Golden_Tenerife_2026();
Golden_Tenerife_low();
Golden_South_2010();
Golden_Dut1();
Golden_HA_Wrap();
Golden_Near_The_Poles();
Golden_Exact_Poles();
Hour_Angle_Is_Periodic();
Longitude_Is_Periodic();
Outputs_Stay_In_Range();
Round_Trip_Through_RADEC2HADEC();
Inputs_Are_Not_Modified();
Cyclic_Calls_With_Inputs_Set_Once_Are_Stable();

METHOD PRIVATE CheckNear
VAR_INPUT
	fExpected	: LREAL;
	fActual	: LREAL;
	fDelta	: LREAL;
	sName	: STRING(255);
END_VAR
AssertEquals_LREAL(Expected := fExpected, Actual := fActual, Delta := fDelta, Message := sName);
END_METHOD

METHOD PRIVATE CheckAngle
VAR_INPUT
	fExpected	: LREAL;
	fActual	: LREAL;
	fDelta	: LREAL;
	sName	: STRING(255);
END_VAR
VAR
	fDiff	: LREAL;
END_VAR
// angles in degrees, compared modulo 360 so that 359.9999999 and -1.0E-7 are equal
fDiff := fActual - fExpected;
WHILE fDiff > 180.0 DO fDiff := fDiff - 360.0; END_WHILE
WHILE fDiff < -180.0 DO fDiff := fDiff + 360.0; END_WHILE
AssertEquals_LREAL(Expected := 0.0, Actual := fDiff, Delta := fDelta, Message := sName);
END_METHOD

METHOD PRIVATE CheckSeparation
VAR_INPUT
	fLon1	: LREAL;
	fLat1	: LREAL;
	fLon2	: LREAL;
	fLat2	: LREAL;
	fDelta	: LREAL;
	sName	: STRING(255);
END_VAR
VAR
	fD2r	: LREAL;
	fHalfDLat	: LREAL;
	fHalfDLon	: LREAL;
	fHav	: LREAL;
	fSep	: LREAL;
END_VAR
// great-circle separation of two positions (longitude, latitude in degrees) against a tolerance in degrees;
// a difference of longitudes is not a distance on the sky, this is (haversine formula)
fD2r := 0.017453292519943295;
fHalfDLat := (fLat2 - fLat1) * fD2r * 0.5;
fHalfDLon := (fLon2 - fLon1) * fD2r * 0.5;
fHav := SIN(fHalfDLat) * SIN(fHalfDLat) + COS(fLat1 * fD2r) * COS(fLat2 * fD2r) * SIN(fHalfDLon) * SIN(fHalfDLon);
fSep := 2.0 * ASIN(SQRT(LIMIT(0.0, fHav, 1.0))) / fD2r;
AssertEquals_LREAL(Expected := 0.0, Actual := fSep, Delta := fDelta, Message := sName);
END_METHOD

METHOD PRIVATE Golden_Tenerife_2026
VAR
	fb	: AstroBROT.FB_HADEC2RADEC;
END_VAR
TEST('Golden_Tenerife_2026');
fb(jd := 2461300.75, ha := 345.0, dec := 22.01, lon := -16.5, dut1 := 0.0);
CheckAngle(84.28759958479777, fb.ra_out, 1.0E-7, 'Tenerife_2026 ra');
CheckNear(21.993212482320583, fb.dec_out, 1.0E-7, 'Tenerife_2026 dec');
CheckSeparation(84.28749809589803, 21.9932192971722, fb.ra_out, fb.dec_out, 0.0002, 'Tenerife_2026 vs erfa');
TEST_FINISHED();
END_METHOD

METHOD PRIVATE Golden_Tenerife_low
VAR
	fb	: AstroBROT.FB_HADEC2RADEC;
END_VAR
TEST('Golden_Tenerife_low');
fb(jd := 2461300.75, ha := 30.0, dec := -10.0, lon := -16.5, dut1 := 0.0);
CheckAngle(39.36056226713681, fb.ra_out, 1.0E-7, 'Tenerife_low ra');
CheckNear(-10.11975028485237, fb.dec_out, 1.0E-7, 'Tenerife_low dec');
CheckSeparation(39.36047119642502, -10.11974494836338, fb.ra_out, fb.dec_out, 0.0002, 'Tenerife_low vs erfa');
TEST_FINISHED();
END_METHOD

METHOD PRIVATE Golden_South_2010
VAR
	fb	: AstroBROT.FB_HADEC2RADEC;
END_VAR
TEST('Golden_South_2010');
fb(jd := 2455197.5, ha := 100.0, dec := -47.3, lon := -70.7, dut1 := 0.0);
CheckAngle(289.6589544745373, fb.ra_out, 1.0E-7, 'South_2010 ra');
CheckNear(-47.317658585279744, fb.dec_out, 1.0E-7, 'South_2010 dec');
CheckSeparation(289.65896142189746, -47.31759859445048, fb.ra_out, fb.dec_out, 0.0002, 'South_2010 vs erfa');
TEST_FINISHED();
END_METHOD

METHOD PRIVATE Golden_Dut1
VAR
	fb	: AstroBROT.FB_HADEC2RADEC;
END_VAR
TEST('Golden_Dut1');
fb(jd := 2461300.75, ha := 345.0, dec := 22.01, lon := -16.5, dut1 := 0.9);
CheckAngle(84.29135982739001, fb.ra_out, 1.0E-7, 'Tenerife_dut1_plus ra');
CheckNear(21.993222245664892, fb.dec_out, 1.0E-7, 'Tenerife_dut1_plus dec');
CheckSeparation(84.2912582746304, 21.993229060334635, fb.ra_out, fb.dec_out, 0.0002, 'Tenerife_dut1_plus vs erfa');
fb(jd := 2461300.75, ha := 345.0, dec := 22.01, lon := -16.5, dut1 := -0.9);
CheckAngle(84.28383934246425, fb.ra_out, 1.0E-7, 'Tenerife_dut1_minus ra');
CheckNear(21.993202719039957, fb.dec_out, 1.0E-7, 'Tenerife_dut1_minus dec');
CheckSeparation(84.28373791742105, 21.993209534073422, fb.ra_out, fb.dec_out, 0.0002, 'Tenerife_dut1_minus vs erfa');
TEST_FINISHED();
END_METHOD

METHOD PRIVATE Golden_HA_Wrap
VAR
	fb	: AstroBROT.FB_HADEC2RADEC;
END_VAR
TEST('Golden_HA_Wrap');
fb(jd := 2461300.75, ha := 0.0001, dec := 22.01, lon := -16.5, dut1 := 0.0);
CheckAngle(69.28989220623771, fb.ra_out, 1.0E-7, 'HA_wrap_low ra');
CheckNear(21.955213314004528, fb.dec_out, 1.0E-7, 'HA_wrap_low dec');
CheckSeparation(69.28978714407457, 21.95521257782602, fb.ra_out, fb.dec_out, 0.0002, 'HA_wrap_low vs erfa');
fb(jd := 2461300.75, ha := 359.9999, dec := 22.01, lon := -16.5, dut1 := 0.0);
CheckAngle(69.29009214752863, fb.ra_out, 1.0E-7, 'HA_wrap_high ra');
CheckNear(21.95521380223834, fb.dec_out, 1.0E-7, 'HA_wrap_high dec');
CheckSeparation(69.28998708537415, 21.955213066161644, fb.ra_out, fb.dec_out, 0.0002, 'HA_wrap_high vs erfa');
TEST_FINISHED();
END_METHOD

METHOD PRIVATE Golden_Near_The_Poles
VAR
	fb	: AstroBROT.FB_HADEC2RADEC;
END_VAR
TEST('Golden_Near_The_Poles');
fb(jd := 2461300.75, ha := 200.0, dec := 89.9, lon := -16.5, dut1 := 0.0);
CheckAngle(316.7079065490832, fb.ra_out, 1.0E-7, 'Near_north_pole ra');
CheckNear(89.8844737036994, fb.dec_out, 1.0E-7, 'Near_north_pole dec');
CheckSeparation(316.7064081660361, 89.88445978947462, fb.ra_out, fb.dec_out, 0.0002, 'Near_north_pole vs erfa');
fb(jd := 2455197.5, ha := 200.0, dec := -89.9, lon := -70.7, dut1 := 0.0);
CheckAngle(186.30600937346122, fb.ra_out, 1.0E-7, 'Near_south_pole ra');
CheckNear(-89.84872530394176, fb.dec_out, 1.0E-7, 'Near_south_pole dec');
CheckSeparation(186.3367115207879, -89.84875262097749, fb.ra_out, fb.dec_out, 0.0002, 'Near_south_pole vs erfa');
TEST_FINISHED();
END_METHOD

METHOD PRIVATE Golden_Exact_Poles
VAR
	fb	: AstroBROT.FB_HADEC2RADEC;
END_VAR
TEST('Golden_Exact_Poles');
fb(jd := 2461300.75, ha := 200.0, dec := 90.0, lon := -16.5, dut1 := 0.0);
// at exactly dec = +-90 neither ra nor dec is reproducible (d_ra ~ 1/cos(dec) = 1E16, and d_dec is evaluated at that ra), only the bound against erfa is pinned
CheckSeparation(358.71048545509177, 89.85071696591022, fb.ra_out, fb.dec_out, 0.015, 'North_pole vs erfa');
fb(jd := 2455197.5, ha := 200.0, dec := -90.0, lon := -70.7, dut1 := 0.0);
// at exactly dec = +-90 neither ra nor dec is reproducible (d_ra ~ 1/cos(dec) = 1E16, and d_dec is evaluated at that ra), only the bound against erfa is pinned
CheckSeparation(179.80951066897055, -89.94824466951559, fb.ra_out, fb.dec_out, 0.015, 'South_pole vs erfa');
TEST_FINISHED();
END_METHOD

METHOD PRIVATE Hour_Angle_Is_Periodic
VAR
	fb	: AstroBROT.FB_HADEC2RADEC;
END_VAR
TEST('Hour_Angle_Is_Periodic');
// ha and ha +- 360 are the same position; the block does not wrap ra before the corrections, so this also covers the wrap of d_ra (issue #10)
fb(jd := 2461300.75, ha := -15.0, dec := 22.01, lon := -16.5);
CheckAngle(84.28759958479777, fb.ra_out, 1.0E-9, 'ha - 360 ra');
CheckNear(21.993212482320583, fb.dec_out, 1.0E-9, 'ha - 360 dec');
fb(jd := 2461300.75, ha := 705.0, dec := 22.01, lon := -16.5);
CheckAngle(84.28759958479777, fb.ra_out, 1.0E-9, 'ha + 360 ra');
CheckNear(21.993212482320583, fb.dec_out, 1.0E-9, 'ha + 360 dec');
AssertTrue(Condition := fb.ra_out >= 0.0 AND fb.ra_out < 360.0, Message := 'ra_out is within 0 <= ra < 360');
TEST_FINISHED();
END_METHOD

METHOD PRIVATE Longitude_Is_Periodic
VAR
	fb	: AstroBROT.FB_HADEC2RADEC;
END_VAR
TEST('Longitude_Is_Periodic');
fb(jd := 2461300.75, ha := 345.0, dec := 22.01, lon := 343.5);
CheckAngle(84.28759958479777, fb.ra_out, 1.0E-9, 'lon + 360 ra');
fb(jd := 2461300.75, ha := 345.0, dec := 22.01, lon := -376.5);
CheckAngle(84.28759958479777, fb.ra_out, 1.0E-9, 'lon - 360 ra');
TEST_FINISHED();
END_METHOD

METHOD PRIVATE Outputs_Stay_In_Range
VAR
	fb	: AstroBROT.FB_HADEC2RADEC;
	i	: INT;
	fHa	: LREAL;
END_VAR
TEST('Outputs_Stay_In_Range');
FOR i := -1 TO 8 DO
	fHa := 45.0 * i;
	fb(jd := 2461300.75, ha := fHa, dec := 89.9, lon := -16.5);
	AssertTrue(Condition := fb.ra_out >= 0.0 AND fb.ra_out < 360.0 AND fb.dec_out <= 90.0 AND fb.dec_out >= -90.0, Message := 'ha sweep at dec +89.9 stays in range');
	fb(jd := 2461300.75, ha := fHa, dec := -89.9, lon := -16.5);
	AssertTrue(Condition := fb.ra_out >= 0.0 AND fb.ra_out < 360.0 AND fb.dec_out <= 90.0 AND fb.dec_out >= -90.0, Message := 'ha sweep at dec -89.9 stays in range');
	fb(jd := 2461300.75, ha := fHa, dec := 0.0, lon := -16.5);
	AssertTrue(Condition := fb.ra_out >= 0.0 AND fb.ra_out < 360.0 AND fb.dec_out <= 90.0 AND fb.dec_out >= -90.0, Message := 'ha sweep at dec 0 stays in range');
END_FOR
TEST_FINISHED();
END_METHOD

METHOD PRIVATE Round_Trip_Through_RADEC2HADEC
VAR
	fbFwd	: AstroBROT.FB_RADEC2HADEC;
	fbBack	: AstroBROT.FB_HADEC2RADEC;
END_VAR
TEST('Round_Trip_Through_RADEC2HADEC');
// the two blocks are only approximate inverses (nutation and aberration are applied at slightly different
// positions), so 1E-6 deg away from the poles and 2E-4 deg (0.72 arcsec) 0.1 deg from a pole
fbFwd(jd := 2461300.75, ra := 83.63, dec := 22.01, lon := -16.5);
fbBack(jd := 2461300.75, ha := fbFwd.ha_out, dec := fbFwd.dec_out, lon := -16.5);
CheckSeparation(83.63, 22.01, fbBack.ra_out, fbBack.dec_out, 1.0E-6, 'Tenerife_2026');
fbFwd(jd := 2455197.5, ra := 312.5, dec := -47.3, lon := -70.7);
fbBack(jd := 2455197.5, ha := fbFwd.ha_out, dec := fbFwd.dec_out, lon := -70.7);
CheckSeparation(312.5, -47.3, fbBack.ra_out, fbBack.dec_out, 1.0E-6, 'South_2010');
fbFwd(jd := 2461300.75, ra := 359.9999, dec := 22.01, lon := -16.5);
fbBack(jd := 2461300.75, ha := fbFwd.ha_out, dec := fbFwd.dec_out, lon := -16.5);
CheckSeparation(359.9999, 22.01, fbBack.ra_out, fbBack.dec_out, 1.0E-6, 'RA just below 360');
fbFwd(jd := 2461300.75, ra := 0.0001, dec := 22.01, lon := -16.5);
fbBack(jd := 2461300.75, ha := fbFwd.ha_out, dec := fbFwd.dec_out, lon := -16.5);
CheckSeparation(0.0001, 22.01, fbBack.ra_out, fbBack.dec_out, 1.0E-6, 'RA just above 0');
fbFwd(jd := 2461300.75, ra := 200.0, dec := 89.9, lon := -16.5);
fbBack(jd := 2461300.75, ha := fbFwd.ha_out, dec := fbFwd.dec_out, lon := -16.5);
CheckSeparation(200.0, 89.9, fbBack.ra_out, fbBack.dec_out, 0.0002, 'near the north pole');
TEST_FINISHED();
END_METHOD

METHOD PRIVATE Inputs_Are_Not_Modified
VAR
	fb	: AstroBROT.FB_HADEC2RADEC;
END_VAR
TEST('Inputs_Are_Not_Modified');
fb(jd := 2461300.75, ha := 345.0, dec := 22.01, lon := -16.5, dut1 := 0.5);
CheckNear(2461300.75, fb.jd, 0.0, 'jd unchanged');
CheckNear(345.0, fb.ha, 0.0, 'ha unchanged');
CheckNear(22.01, fb.dec, 0.0, 'dec unchanged');
CheckNear(-16.5, fb.lon, 0.0, 'lon unchanged');
CheckNear(0.5, fb.dut1, 0.0, 'dut1 unchanged');
TEST_FINISHED();
END_METHOD

METHOD PRIVATE Cyclic_Calls_With_Inputs_Set_Once_Are_Stable
VAR
	fb	: AstroBROT.FB_HADEC2RADEC;
	i	: INT;
END_VAR
TEST('Cyclic_Calls_With_Inputs_Set_Once_Are_Stable');
fb.jd := 2461300.75;
fb.ha := 345.0;
fb.dec := 22.01;
fb.lon := -16.5;
FOR i := 1 TO 5 DO
	fb();
	CheckAngle(84.28759958479777, fb.ra_out, 1.0E-7, 'cyclic call ra');
	CheckNear(21.993212482320583, fb.dec_out, 1.0E-7, 'cyclic call dec');
END_FOR
TEST_FINISHED();
END_METHOD

END_FUNCTION_BLOCK

// ---- POUs/FB_SUNPOS_Tests.TcPOU
// Tests for AstroBROT.FB_SUNPOS (apparent position of the Sun, port of IDLAstro sunpos.pro).
//
// GENERATED by AstroBROT/testing/gen_block_tests.py from testing/golden_blocks.py, do not edit the numbers by hand.
// Golden values from the Python port of the ST (1E-7 deg). Independently of the port the position is compared with a
// position built from erfa (epv00 / pmat06 / nut06a): 1.5E-3 deg = 5.4 arcsec, the measured maximum is 3.2 arcsec and
// the IDLAstro documentation states 7.3 arcsec for 1900-2100. The last tests are plain sanity checks (equinox,
// solstice, obliquity, RA rate) that need neither the port nor erfa.
FUNCTION_BLOCK FB_SUNPOS_Tests EXTENDS TcUnit.FB_TestSuite
VAR
END_VAR

Golden_Epoch_1900_And_J2000();
Golden_Start_2010();
Golden_Tenerife_2026();
Golden_Year_2050();
Golden_Equinox_And_Solstice_2026();
Sanity_Equinox_Solstice_Obliquity();
Sanity_Right_Ascension_Advances_About_One_Degree_Per_Day();
Inputs_Are_Not_Modified();
Cyclic_Calls_With_Inputs_Set_Once_Are_Stable();

METHOD PRIVATE CheckNear
VAR_INPUT
	fExpected	: LREAL;
	fActual	: LREAL;
	fDelta	: LREAL;
	sName	: STRING(255);
END_VAR
AssertEquals_LREAL(Expected := fExpected, Actual := fActual, Delta := fDelta, Message := sName);
END_METHOD

METHOD PRIVATE CheckAngle
VAR_INPUT
	fExpected	: LREAL;
	fActual	: LREAL;
	fDelta	: LREAL;
	sName	: STRING(255);
END_VAR
VAR
	fDiff	: LREAL;
END_VAR
// angles in degrees, compared modulo 360 so that 359.9999999 and -1.0E-7 are equal
fDiff := fActual - fExpected;
WHILE fDiff > 180.0 DO fDiff := fDiff - 360.0; END_WHILE
WHILE fDiff < -180.0 DO fDiff := fDiff + 360.0; END_WHILE
AssertEquals_LREAL(Expected := 0.0, Actual := fDiff, Delta := fDelta, Message := sName);
END_METHOD

METHOD PRIVATE CheckSeparation
VAR_INPUT
	fLon1	: LREAL;
	fLat1	: LREAL;
	fLon2	: LREAL;
	fLat2	: LREAL;
	fDelta	: LREAL;
	sName	: STRING(255);
END_VAR
VAR
	fD2r	: LREAL;
	fHalfDLat	: LREAL;
	fHalfDLon	: LREAL;
	fHav	: LREAL;
	fSep	: LREAL;
END_VAR
// great-circle separation of two positions (longitude, latitude in degrees) against a tolerance in degrees;
// a difference of longitudes is not a distance on the sky, this is (haversine formula)
fD2r := 0.017453292519943295;
fHalfDLat := (fLat2 - fLat1) * fD2r * 0.5;
fHalfDLon := (fLon2 - fLon1) * fD2r * 0.5;
fHav := SIN(fHalfDLat) * SIN(fHalfDLat) + COS(fLat1 * fD2r) * COS(fLat2 * fD2r) * SIN(fHalfDLon) * SIN(fHalfDLon);
fSep := 2.0 * ASIN(SQRT(LIMIT(0.0, fHav, 1.0))) / fD2r;
AssertEquals_LREAL(Expected := 0.0, Actual := fSep, Delta := fDelta, Message := sName);
END_METHOD

METHOD PRIVATE Golden_Epoch_1900_And_J2000
VAR
	fb	: AstroBROT.FB_SUNPOS;
END_VAR
TEST('Golden_Epoch_1900_And_J2000');
fb(jd := 2415020.0);
CheckAngle(280.4932027906667, fb.ra, 1.0E-7, 'Epoch_1900 ra');
CheckNear(-23.1010537507843, fb.dec, 1.0E-7, 'Epoch_1900 dec');
CheckNear(279.6444003923051, fb.longmed, 1.0E-7, 'Epoch_1900 longmed');
CheckNear(23.451814403891508, fb.oblt, 1.0E-7, 'Epoch_1900 oblt');
CheckSeparation(280.49336588705194, -23.100882447052207, fb.ra, fb.dec, 0.0015, 'Epoch_1900 vs erfa');
fb(jd := 2451545.0);
CheckAngle(281.27675114506104, fb.ra, 1.0E-7, 'J2000 ra');
CheckNear(-23.03291144063576, fb.dec, 1.0E-7, 'J2000 dec');
CheckNear(280.37698786565545, fb.longmed, 1.0E-7, 'J2000 longmed');
CheckNear(23.437814186179185, fb.oblt, 1.0E-7, 'J2000 oblt');
CheckSeparation(281.2776898567173, -23.032708521099703, fb.ra, fb.dec, 0.0015, 'J2000 vs erfa');
TEST_FINISHED();
END_METHOD

METHOD PRIVATE Golden_Start_2010
VAR
	fb	: AstroBROT.FB_SUNPOS;
END_VAR
TEST('Golden_Start_2010');
fb(jd := 2455197.5);
CheckAngle(281.36670259981736, fb.ra, 1.0E-7, 'Start_2010 ra');
CheckNear(-23.027520406003863, fb.dec, 1.0E-7, 'Start_2010 dec');
CheckNear(280.4515850797381, fb.longmed, 1.0E-7, 'Start_2010 longmed');
CheckNear(23.438922135094707, fb.oblt, 1.0E-7, 'Start_2010 oblt');
CheckSeparation(281.3668435021951, -23.027353107638568, fb.ra, fb.dec, 0.0015, 'Start_2010 vs erfa');
TEST_FINISHED();
END_METHOD

METHOD PRIVATE Golden_Tenerife_2026
VAR
	fb	: AstroBROT.FB_SUNPOS;
END_VAR
TEST('Golden_Tenerife_2026');
fb(jd := 2461300.75);
CheckAngle(174.8393337772982, fb.ra, 1.0E-7, 'Tenerife_2026 ra');
CheckNear(2.2331274030840897, fb.dec, 1.0E-7, 'Tenerife_2026 dec');
CheckNear(174.38128640738705, fb.longmed, 1.0E-7, 'Tenerife_2026 longmed');
CheckNear(23.437983366242445, fb.oblt, 1.0E-7, 'Tenerife_2026 oblt');
CheckSeparation(174.84005201634432, 2.232830546071217, fb.ra, fb.dec, 0.0015, 'Tenerife_2026 vs erfa');
TEST_FINISHED();
END_METHOD

METHOD PRIVATE Golden_Year_2050
VAR
	fb	: AstroBROT.FB_SUNPOS;
END_VAR
TEST('Golden_Year_2050');
fb(jd := 2469807.5);
CheckAngle(281.68738605381645, fb.ra, 1.0E-7, 'Year_2050 ra');
CheckNear(-22.996590225692305, fb.dec, 1.0E-7, 'Year_2050 dec');
CheckNear(280.748664812077, fb.longmed, 1.0E-7, 'Year_2050 longmed');
CheckNear(23.431419887249728, fb.oblt, 1.0E-7, 'Year_2050 oblt');
CheckSeparation(281.6880601925095, -22.996415910571415, fb.ra, fb.dec, 0.0015, 'Year_2050 vs erfa');
TEST_FINISHED();
END_METHOD

METHOD PRIVATE Golden_Equinox_And_Solstice_2026
VAR
	fb	: AstroBROT.FB_SUNPOS;
END_VAR
TEST('Golden_Equinox_And_Solstice_2026');
fb(jd := 2461120.5);
CheckAngle(0.3503559250411667, fb.ra, 1.0E-7, 'March_equinox_2026 ra');
CheckNear(0.15188894029624206, fb.dec, 1.0E-7, 'March_equinox_2026 dec');
CheckNear(0.3857660381664108, fb.longmed, 1.0E-7, 'March_equinox_2026 longmed');
CheckNear(23.438239257244735, fb.oblt, 1.0E-7, 'March_equinox_2026 oblt');
CheckSeparation(0.35013805050580776, 0.15179565874940165, fb.ra, fb.dec, 0.0015, 'March_equinox_2026 vs erfa');
fb(jd := 2461212.5);
CheckAngle(89.63389115907498, fb.ra, 1.0E-7, 'June_solstice_2026 ra');
CheckNear(23.437689690338015, fb.dec, 1.0E-7, 'June_solstice_2026 dec');
CheckNear(89.66763149502222, fb.longmed, 1.0E-7, 'June_solstice_2026 longmed');
CheckNear(23.43811655330089, fb.oblt, 1.0E-7, 'June_solstice_2026 oblt');
CheckSeparation(89.63460394632473, 23.437550528896672, fb.ra, fb.dec, 0.0015, 'June_solstice_2026 vs erfa');
TEST_FINISHED();
END_METHOD

METHOD PRIVATE Sanity_Equinox_Solstice_Obliquity
VAR
	fb	: AstroBROT.FB_SUNPOS;
END_VAR
TEST('Sanity_Equinox_Solstice_Obliquity');
// 2026-03-21 00:00 UT is 9 h after the March equinox: the Sun is at RA about 0.35 deg, Dec about +0.15 deg
fb(jd := 2461120.5);
CheckAngle(0.35, fb.ra, 0.3, 'March equinox ra');
CheckNear(0.15, fb.dec, 0.1, 'March equinox dec');
// 2026-06-21 00:00 UT is 8 h before the June solstice: Dec is at its maximum, RA about 89.6 deg
fb(jd := 2461212.5);
CheckNear(23.44, fb.dec, 0.02, 'June solstice dec');
CheckAngle(89.6, fb.ra, 0.3, 'June solstice ra');
// true obliquity of the ecliptic in 2026
CheckNear(23.437, fb.oblt, 0.005, 'oblt 2026');
TEST_FINISHED();
END_METHOD

METHOD PRIVATE Sanity_Right_Ascension_Advances_About_One_Degree_Per_Day
VAR
	fb	: AstroBROT.FB_SUNPOS;
	fbNext	: AstroBROT.FB_SUNPOS;
	i	: INT;
	fStep	: LREAL;
END_VAR
TEST('Sanity_Right_Ascension_Advances_About_One_Degree_Per_Day');
// over a year the daily change of RA is between 0.85 and 1.15 deg (0.91 to 1.11 in reality); this also crosses the wrap at 360
FOR i := 0 TO 36 DO
	fb(jd := 2461041.5 + 10.0 * i);
	fbNext(jd := 2461042.5 + 10.0 * i);
	fStep := fbNext.ra - fb.ra;
	IF fStep < 0.0 THEN fStep := fStep + 360.0; END_IF
	AssertTrue(Condition := fStep > 0.85 AND fStep < 1.15, Message := 'daily RA step within 0.85 .. 1.15 deg');
	AssertTrue(Condition := fb.ra >= 0.0 AND fb.ra < 360.0 AND ABS(fb.dec) < 23.5, Message := 'ra in range, |dec| below the obliquity');
END_FOR
TEST_FINISHED();
END_METHOD

METHOD PRIVATE Inputs_Are_Not_Modified
VAR
	fb	: AstroBROT.FB_SUNPOS;
END_VAR
TEST('Inputs_Are_Not_Modified');
fb(jd := 2461300.75);
CheckNear(2461300.75, fb.jd, 0.0, 'jd unchanged');
TEST_FINISHED();
END_METHOD

METHOD PRIVATE Cyclic_Calls_With_Inputs_Set_Once_Are_Stable
VAR
	fb	: AstroBROT.FB_SUNPOS;
	i	: INT;
END_VAR
TEST('Cyclic_Calls_With_Inputs_Set_Once_Are_Stable');
fb.jd := 2461300.75;
FOR i := 1 TO 5 DO
	fb();
	CheckAngle(174.8393337772982, fb.ra, 1.0E-7, 'cyclic call ra');
	CheckNear(2.2331274030840897, fb.dec, 1.0E-7, 'cyclic call dec');
END_FOR
TEST_FINISHED();
END_METHOD

END_FUNCTION_BLOCK

// ---- POUs/FB_EdgeCases_Tests.TcPOU
// Edge cases of FB_EQ2HOR and FB_HOR2EQ: the celestial poles, an observer at a pole and on the equator, the zenith and
// the nadir, wrap-around of RA and azimuth, positions below the horizon and out-of-range angles.
//
// GENERATED by AstroBROT/testing/gen_block_tests.py from testing/golden_blocks.py, do not edit the numbers by hand.
// Every golden case is checked against the Python port of the ST (1E-7 deg) and against erfa (atco13 / atoc13) as a
// great-circle separation (2E-4 deg = 0.72 arcsec, no refraction, dut1 = 0). Altitude and azimuth are compared as a
// separation on the sky, not as two separate angle differences: near the zenith an azimuth difference is amplified by
// 1 / cos(alt) and says little about the pointing error (Azimuth_Difference_Is_Not_A_Sky_Separation).
FUNCTION_BLOCK FB_EdgeCases_Tests EXTENDS TcUnit.FB_TestSuite
VAR
END_VAR

EQ2HOR_North_celestial_pole();
EQ2HOR_South_celestial_pole();
EQ2HOR_RA_wrap_low();
EQ2HOR_RA_wrap_high();
EQ2HOR_Below_horizon();
EQ2HOR_Observer_at_north_pole();
EQ2HOR_Observer_at_south_pole();
EQ2HOR_Observer_on_equator();
HOR2EQ_Zenith_az0();
HOR2EQ_Zenith_az180();
HOR2EQ_Nadir();
HOR2EQ_Horizon_north();
HOR2EQ_Az_wrap_low();
HOR2EQ_Az_wrap_high();
HOR2EQ_Observer_at_north_pole();
HOR2EQ_Observer_at_south_pole();
HOR2EQ_Observer_on_equator();
HOR2EQ_Azimuth_Does_Not_Matter_At_The_Zenith();
HOR2EQ_Azimuth_Is_Periodic();
EQ2HOR_Right_Ascension_Is_Periodic();
EQ2HOR_Longitude_Is_Periodic();
EQ2HOR_Outputs_Stay_In_Range();
HOR2EQ_Outputs_Stay_In_Range();
Azimuth_Difference_Is_Not_A_Sky_Separation();

METHOD PRIVATE CheckNear
VAR_INPUT
	fExpected	: LREAL;
	fActual	: LREAL;
	fDelta	: LREAL;
	sName	: STRING(255);
END_VAR
AssertEquals_LREAL(Expected := fExpected, Actual := fActual, Delta := fDelta, Message := sName);
END_METHOD

METHOD PRIVATE CheckAngle
VAR_INPUT
	fExpected	: LREAL;
	fActual	: LREAL;
	fDelta	: LREAL;
	sName	: STRING(255);
END_VAR
VAR
	fDiff	: LREAL;
END_VAR
// angles in degrees, compared modulo 360 so that 359.9999999 and -1.0E-7 are equal
fDiff := fActual - fExpected;
WHILE fDiff > 180.0 DO fDiff := fDiff - 360.0; END_WHILE
WHILE fDiff < -180.0 DO fDiff := fDiff + 360.0; END_WHILE
AssertEquals_LREAL(Expected := 0.0, Actual := fDiff, Delta := fDelta, Message := sName);
END_METHOD

METHOD PRIVATE CheckSeparation
VAR_INPUT
	fLon1	: LREAL;
	fLat1	: LREAL;
	fLon2	: LREAL;
	fLat2	: LREAL;
	fDelta	: LREAL;
	sName	: STRING(255);
END_VAR
VAR
	fD2r	: LREAL;
	fHalfDLat	: LREAL;
	fHalfDLon	: LREAL;
	fHav	: LREAL;
	fSep	: LREAL;
END_VAR
// great-circle separation of two positions (longitude, latitude in degrees) against a tolerance in degrees;
// a difference of longitudes is not a distance on the sky, this is (haversine formula)
fD2r := 0.017453292519943295;
fHalfDLat := (fLat2 - fLat1) * fD2r * 0.5;
fHalfDLon := (fLon2 - fLon1) * fD2r * 0.5;
fHav := SIN(fHalfDLat) * SIN(fHalfDLat) + COS(fLat1 * fD2r) * COS(fLat2 * fD2r) * SIN(fHalfDLon) * SIN(fHalfDLon);
fSep := 2.0 * ASIN(SQRT(LIMIT(0.0, fHav, 1.0))) / fD2r;
AssertEquals_LREAL(Expected := 0.0, Actual := fSep, Delta := fDelta, Message := sName);
END_METHOD

METHOD PRIVATE EQ2HOR_North_celestial_pole
VAR
	fb	: AstroBROT.FB_EQ2HOR;
END_VAR
TEST('EQ2HOR_North_celestial_pole');
fb(ra := 0.0, dec := 90.0, jd := 2461300.75, lon := -16.5, lat := 28.3, refract := FALSE);
CheckNear(28.250439967419368, fb.alt, 1.0E-7, 'North_celestial_pole alt');
CheckAngle(0.15978772490399448, fb.az, 1.0E-7, 'North_celestial_pole az');
CheckSeparation(0.159877225222193, 28.250414281534653, fb.az, fb.alt, 0.0002, 'North_celestial_pole vs erfa');
TEST_FINISHED();
END_METHOD

METHOD PRIVATE EQ2HOR_South_celestial_pole
VAR
	fb	: AstroBROT.FB_EQ2HOR;
END_VAR
TEST('EQ2HOR_South_celestial_pole');
fb(ra := 0.0, dec := -90.0, jd := 2455197.5, lon := -70.7, lat := -30.2, refract := FALSE);
CheckNear(30.24486015624291, fb.alt, 1.0E-7, 'South_celestial_pole alt');
CheckAngle(180.02996665539834, fb.az, 1.0E-7, 'South_celestial_pole az');
CheckSeparation(180.02986430898196, 30.244862822992012, fb.az, fb.alt, 0.0002, 'South_celestial_pole vs erfa');
TEST_FINISHED();
END_METHOD

METHOD PRIVATE EQ2HOR_RA_wrap_low
VAR
	fb	: AstroBROT.FB_EQ2HOR;
END_VAR
TEST('EQ2HOR_RA_wrap_low');
fb(ra := 0.0001, dec := 22.01, jd := 2461300.75, lon := -16.5, lat := 28.3, refract := FALSE);
CheckNear(27.80734764100336, fb.alt, 1.0E-7, 'RA_wrap_low alt');
CheckAngle(281.5592750159755, fb.az, 1.0E-7, 'RA_wrap_low az');
CheckSeparation(281.55928456225905, 27.807403036183125, fb.az, fb.alt, 0.0002, 'RA_wrap_low vs erfa');
TEST_FINISHED();
END_METHOD

METHOD PRIVATE EQ2HOR_RA_wrap_high
VAR
	fb	: AstroBROT.FB_EQ2HOR;
END_VAR
TEST('EQ2HOR_RA_wrap_high');
fb(ra := 359.9999, dec := 22.01, jd := 2461300.75, lon := -16.5, lat := 28.3, refract := FALSE);
CheckNear(27.807174935931986, fb.alt, 1.0E-7, 'RA_wrap_high alt');
CheckAngle(281.55935130398774, fb.az, 1.0E-7, 'RA_wrap_high az');
CheckSeparation(281.5593608503559, 27.80723033089579, fb.az, fb.alt, 0.0002, 'RA_wrap_high vs erfa');
TEST_FINISHED();
END_METHOD

METHOD PRIVATE EQ2HOR_Below_horizon
VAR
	fb	: AstroBROT.FB_EQ2HOR;
END_VAR
TEST('EQ2HOR_Below_horizon');
fb(ra := 200.0, dec := -60.0, jd := 2461300.75, lon := -16.5, lat := 28.3, refract := FALSE);
CheckNear(-44.20054793244784, fb.alt, 1.0E-7, 'Below_horizon alt');
CheckAngle(148.24726062401623, fb.az, 1.0E-7, 'Below_horizon az');
CheckSeparation(148.2471745159021, -44.20052670358075, fb.az, fb.alt, 0.0002, 'Below_horizon vs erfa');
TEST_FINISHED();
END_METHOD

METHOD PRIVATE EQ2HOR_Observer_at_north_pole
VAR
	fb	: AstroBROT.FB_EQ2HOR;
END_VAR
TEST('EQ2HOR_Observer_at_north_pole');
fb(ra := 83.63, dec := 22.01, jd := 2461300.75, lon := 0.0, lat := 90.0, refract := FALSE);
CheckNear(22.028492329681235, fb.alt, 1.0E-7, 'Observer_at_north_pole alt');
CheckAngle(182.15756303104874, fb.az, 1.0E-7, 'Observer_at_north_pole az');
CheckSeparation(182.15754329791073, 22.028492563126676, fb.az, fb.alt, 0.0002, 'Observer_at_north_pole vs erfa');
TEST_FINISHED();
END_METHOD

METHOD PRIVATE EQ2HOR_Observer_at_south_pole
VAR
	fb	: AstroBROT.FB_EQ2HOR;
END_VAR
TEST('EQ2HOR_Observer_at_south_pole');
fb(ra := 83.63, dec := -22.01, jd := 2461300.75, lon := 0.0, lat := -90.0, refract := FALSE);
CheckNear(21.987455170067353, fb.alt, 1.0E-7, 'Observer_at_south_pole alt');
CheckAngle(357.7223600600331, fb.az, 1.0E-7, 'Observer_at_south_pole az');
CheckSeparation(357.7223798312026, 21.987453746489294, fb.az, fb.alt, 0.0002, 'Observer_at_south_pole vs erfa');
TEST_FINISHED();
END_METHOD

METHOD PRIVATE EQ2HOR_Observer_on_equator
VAR
	fb	: AstroBROT.FB_EQ2HOR;
END_VAR
TEST('EQ2HOR_Observer_on_equator');
fb(ra := 83.63, dec := 22.01, jd := 2461300.75, lon := -16.5, lat := 0.0, refract := FALSE);
CheckNear(63.91012183292501, fb.alt, 1.0E-7, 'Observer_on_equator alt');
CheckAngle(31.47678113024893, fb.az, 1.0E-7, 'Observer_on_equator az');
CheckSeparation(31.476987570998272, 63.910069653766755, fb.az, fb.alt, 0.0002, 'Observer_on_equator vs erfa');
TEST_FINISHED();
END_METHOD

METHOD PRIVATE HOR2EQ_Zenith_az0
VAR
	fb	: AstroBROT.FB_HOR2EQ;
END_VAR
TEST('HOR2EQ_Zenith_az0');
fb(alt := 90.0, az := 0.0, jd := 2461300.75, lon := -16.5, lat := 28.3, refract := FALSE);
CheckAngle(69.27121990661907, fb.ra, 1.0E-7, 'Zenith_az0 ra');
CheckNear(28.245793686130707, fb.dec, 1.0E-7, 'Zenith_az0 dec');
CheckSeparation(69.27111043655914, 28.245793175984534, fb.ra, fb.dec, 0.0002, 'Zenith_az0 vs erfa');
TEST_FINISHED();
END_METHOD

METHOD PRIVATE HOR2EQ_Zenith_az180
VAR
	fb	: AstroBROT.FB_HOR2EQ;
END_VAR
TEST('HOR2EQ_Zenith_az180');
fb(alt := 90.0, az := 180.0, jd := 2461300.75, lon := -16.5, lat := 28.3, refract := FALSE);
CheckAngle(69.27121990661907, fb.ra, 1.0E-7, 'Zenith_az180 ra');
CheckNear(28.245793686130707, fb.dec, 1.0E-7, 'Zenith_az180 dec');
CheckSeparation(69.27111043655914, 28.245793175984534, fb.ra, fb.dec, 0.0002, 'Zenith_az180 vs erfa');
TEST_FINISHED();
END_METHOD

METHOD PRIVATE HOR2EQ_Nadir
VAR
	fb	: AstroBROT.FB_HOR2EQ;
END_VAR
TEST('HOR2EQ_Nadir');
fb(alt := -90.0, az := 0.0, jd := 2461300.75, lon := -16.5, lat := 28.3, refract := FALSE);
CheckAngle(249.2743126674054, fb.ra, 1.0E-7, 'Nadir ra');
CheckNear(-28.244996713786396, fb.dec, 1.0E-7, 'Nadir dec');
CheckSeparation(249.27437964349747, -28.24499592575831, fb.ra, fb.dec, 0.0002, 'Nadir vs erfa');
TEST_FINISHED();
END_METHOD

METHOD PRIVATE HOR2EQ_Horizon_north
VAR
	fb	: AstroBROT.FB_HOR2EQ;
END_VAR
TEST('HOR2EQ_Horizon_north');
fb(alt := 0.0, az := 0.0, jd := 2461300.75, lon := -16.5, lat := 28.3, refract := FALSE);
CheckAngle(249.60995502319435, fb.ra, 1.0E-7, 'Horizon_north ra');
CheckNear(61.7487089558397, fb.dec, 1.0E-7, 'Horizon_north dec');
CheckSeparation(249.61009729239348, 61.74870711776769, fb.ra, fb.dec, 0.0002, 'Horizon_north vs erfa');
TEST_FINISHED();
END_METHOD

METHOD PRIVATE HOR2EQ_Az_wrap_low
VAR
	fb	: AstroBROT.FB_HOR2EQ;
END_VAR
TEST('HOR2EQ_Az_wrap_low');
fb(alt := 45.0, az := 0.0001, jd := 2461300.75, lon := -16.5, lat := 28.3, refract := FALSE);
CheckAngle(68.88002145549598, fb.ra, 1.0E-7, 'Az_wrap_low ra');
CheckNear(73.24907291497094, fb.dec, 1.0E-7, 'Az_wrap_low dec');
CheckSeparation(68.8797303761049, 73.24907332545713, fb.ra, fb.dec, 0.0002, 'Az_wrap_low vs erfa');
TEST_FINISHED();
END_METHOD

METHOD PRIVATE HOR2EQ_Az_wrap_high
VAR
	fb	: AstroBROT.FB_HOR2EQ;
END_VAR
TEST('HOR2EQ_Az_wrap_high');
fb(alt := 45.0, az := 359.9999, jd := 2461300.75, lon := -16.5, lat := 28.3, refract := FALSE);
CheckAngle(68.87953075699878, fb.ra, 1.0E-7, 'Az_wrap_high ra');
CheckNear(73.24907170989893, fb.dec, 1.0E-7, 'Az_wrap_high dec');
CheckSeparation(68.87923967758073, 73.2490721197454, fb.ra, fb.dec, 0.0002, 'Az_wrap_high vs erfa');
TEST_FINISHED();
END_METHOD

METHOD PRIVATE HOR2EQ_Observer_at_north_pole
VAR
	fb	: AstroBROT.FB_HOR2EQ;
END_VAR
TEST('HOR2EQ_Observer_at_north_pole');
fb(alt := 40.0, az := 100.0, jd := 2461300.75, lon := 0.0, lat := 90.0, refract := FALSE);
CheckAngle(165.82212182028053, fb.ra, 1.0E-7, 'Observer_at_north_pole ra');
CheckNear(40.14345354944047, fb.dec, 1.0E-7, 'Observer_at_north_pole dec');
CheckSeparation(165.82210357343894, 40.14345009010985, fb.ra, fb.dec, 0.0002, 'Observer_at_north_pole vs erfa');
TEST_FINISHED();
END_METHOD

METHOD PRIVATE HOR2EQ_Observer_at_south_pole
VAR
	fb	: AstroBROT.FB_HOR2EQ;
END_VAR
TEST('HOR2EQ_Observer_at_south_pole');
fb(alt := -20.0, az := 100.0, jd := 2461300.75, lon := 0.0, lat := -90.0, refract := FALSE);
CheckAngle(185.85805478189764, fb.ra, 1.0E-7, 'Observer_at_south_pole ra');
CheckNear(20.14661753333691, fb.dec, 1.0E-7, 'Observer_at_south_pole dec');
CheckSeparation(185.85803179512064, 20.146612025652036, fb.ra, fb.dec, 0.0002, 'Observer_at_south_pole vs erfa');
TEST_FINISHED();
END_METHOD

METHOD PRIVATE HOR2EQ_Observer_on_equator
VAR
	fb	: AstroBROT.FB_HOR2EQ;
END_VAR
TEST('HOR2EQ_Observer_on_equator');
fb(alt := 60.0, az := 250.0, jd := 2461300.75, lon := -16.5, lat := 0.0, refract := FALSE);
CheckAngle(40.87970090453398, fb.ra, 1.0E-7, 'Observer_on_equator ra');
CheckNear(-9.963791072363595, fb.dec, 1.0E-7, 'Observer_on_equator dec');
CheckSeparation(40.879599464361846, -9.963785329026702, fb.ra, fb.dec, 0.0002, 'Observer_on_equator vs erfa');
TEST_FINISHED();
END_METHOD

METHOD PRIVATE HOR2EQ_Azimuth_Does_Not_Matter_At_The_Zenith
VAR
	fbA	: AstroBROT.FB_HOR2EQ;
	fbB	: AstroBROT.FB_HOR2EQ;
END_VAR
TEST('HOR2EQ_Azimuth_Does_Not_Matter_At_The_Zenith');
fbA(alt := 90.0, az := 0.0, jd := 2461300.75, lon := -16.5, lat := 28.3, refract := FALSE);
fbB(alt := 90.0, az := 180.0, jd := 2461300.75, lon := -16.5, lat := 28.3, refract := FALSE);
CheckAngle(fbA.ra, fbB.ra, 1.0E-9, 'ra');
CheckNear(fbA.dec, fbB.dec, 1.0E-9, 'dec');
AssertTrue(Condition := fbA.dec > 0.0 AND fbA.dec < 90.0, Message := 'the zenith of a northern site has 0 < dec < 90 (no NaN from ASIN)');
TEST_FINISHED();
END_METHOD

METHOD PRIVATE HOR2EQ_Azimuth_Is_Periodic
VAR
	fbRef	: AstroBROT.FB_HOR2EQ;
	fb	: AstroBROT.FB_HOR2EQ;
END_VAR
TEST('HOR2EQ_Azimuth_Is_Periodic');
fbRef(alt := 45.0, az := 350.0, jd := 2461300.75, lon := -16.5, lat := 28.3, refract := FALSE);
fb(alt := 45.0, az := -10.0, jd := 2461300.75, lon := -16.5, lat := 28.3, refract := FALSE);
CheckAngle(fbRef.ra, fb.ra, 1.0E-9, 'az -10 ra');
CheckNear(fbRef.dec, fb.dec, 1.0E-9, 'az -10 dec');
fb(alt := 45.0, az := 710.0, jd := 2461300.75, lon := -16.5, lat := 28.3, refract := FALSE);
CheckAngle(fbRef.ra, fb.ra, 1.0E-9, 'az 710 ra');
CheckNear(fbRef.dec, fb.dec, 1.0E-9, 'az 710 dec');
TEST_FINISHED();
END_METHOD

METHOD PRIVATE EQ2HOR_Right_Ascension_Is_Periodic
VAR
	fbRef	: AstroBROT.FB_EQ2HOR;
	fb	: AstroBROT.FB_EQ2HOR;
END_VAR
TEST('EQ2HOR_Right_Ascension_Is_Periodic');
fbRef(ra := 83.63, dec := 22.01, jd := 2461300.75, lon := -16.5, lat := 28.3, refract := FALSE);
fb(ra := -276.37, dec := 22.01, jd := 2461300.75, lon := -16.5, lat := 28.3, refract := FALSE);
CheckNear(fbRef.alt, fb.alt, 1.0E-9, 'ra -276.37 alt');
CheckAngle(fbRef.az, fb.az, 1.0E-9, 'ra -276.37 az');
fb(ra := 443.63, dec := 22.01, jd := 2461300.75, lon := -16.5, lat := 28.3, refract := FALSE);
CheckNear(fbRef.alt, fb.alt, 1.0E-9, 'ra 443.63 alt');
CheckAngle(fbRef.az, fb.az, 1.0E-9, 'ra 443.63 az');
TEST_FINISHED();
END_METHOD

METHOD PRIVATE EQ2HOR_Longitude_Is_Periodic
VAR
	fbRef	: AstroBROT.FB_EQ2HOR;
	fb	: AstroBROT.FB_EQ2HOR;
END_VAR
TEST('EQ2HOR_Longitude_Is_Periodic');
fbRef(ra := 83.63, dec := 22.01, jd := 2461300.75, lon := -16.5, lat := 28.3, refract := FALSE);
fb(ra := 83.63, dec := 22.01, jd := 2461300.75, lon := 343.5, lat := 28.3, refract := FALSE);
CheckNear(fbRef.alt, fb.alt, 1.0E-9, 'lon 343.5 alt');
CheckAngle(fbRef.az, fb.az, 1.0E-9, 'lon 343.5 az');
TEST_FINISHED();
END_METHOD

METHOD PRIVATE EQ2HOR_Outputs_Stay_In_Range
VAR
	fb	: AstroBROT.FB_EQ2HOR;
	i	: INT;
	fDec	: LREAL;
END_VAR
TEST('EQ2HOR_Outputs_Stay_In_Range');
// declinations from pole to pole for observers at both poles, on the equator and at a mid latitude
FOR i := -2 TO 2 DO
	fDec := 45.0 * i;
	fb(ra := 200.0, dec := fDec, jd := 2461300.75, lon := 0.0, lat := 90.0, refract := FALSE);
	AssertTrue(Condition := fb.alt >= -90.0 AND fb.alt <= 90.0 AND fb.az >= 0.0 AND fb.az <= 360.0, Message := 'observer at the north pole');
	fb(ra := 200.0, dec := fDec, jd := 2461300.75, lon := 0.0, lat := -90.0, refract := FALSE);
	AssertTrue(Condition := fb.alt >= -90.0 AND fb.alt <= 90.0 AND fb.az >= 0.0 AND fb.az <= 360.0, Message := 'observer at the south pole');
	fb(ra := 200.0, dec := fDec, jd := 2461300.75, lon := 0.0, lat := 0.0, refract := FALSE);
	AssertTrue(Condition := fb.alt >= -90.0 AND fb.alt <= 90.0 AND fb.az >= 0.0 AND fb.az <= 360.0, Message := 'observer on the equator');
	fb(ra := 200.0, dec := fDec, jd := 2461300.75, lon := -16.5, lat := 28.3, refract := FALSE);
	AssertTrue(Condition := fb.alt >= -90.0 AND fb.alt <= 90.0 AND fb.az >= 0.0 AND fb.az <= 360.0, Message := 'observer at 28.3 deg');
END_FOR
TEST_FINISHED();
END_METHOD

METHOD PRIVATE HOR2EQ_Outputs_Stay_In_Range
VAR
	fb	: AstroBROT.FB_HOR2EQ;
	i	: INT;
	fAlt	: LREAL;
END_VAR
TEST('HOR2EQ_Outputs_Stay_In_Range');
// altitudes from nadir to zenith, for observers at both poles, on the equator and at a mid latitude
FOR i := -2 TO 2 DO
	fAlt := 45.0 * i;
	fb(alt := fAlt, az := 100.0, jd := 2461300.75, lon := 0.0, lat := 90.0, refract := FALSE);
	AssertTrue(Condition := fb.dec >= -90.0 AND fb.dec <= 90.0 AND fb.ra >= 0.0 AND fb.ra < 360.0, Message := 'observer at the north pole');
	fb(alt := fAlt, az := 100.0, jd := 2461300.75, lon := 0.0, lat := -90.0, refract := FALSE);
	AssertTrue(Condition := fb.dec >= -90.0 AND fb.dec <= 90.0 AND fb.ra >= 0.0 AND fb.ra < 360.0, Message := 'observer at the south pole');
	fb(alt := fAlt, az := 100.0, jd := 2461300.75, lon := 0.0, lat := 0.0, refract := FALSE);
	AssertTrue(Condition := fb.dec >= -90.0 AND fb.dec <= 90.0 AND fb.ra >= 0.0 AND fb.ra < 360.0, Message := 'observer on the equator');
	fb(alt := fAlt, az := 100.0, jd := 2461300.75, lon := -16.5, lat := 28.3, refract := FALSE);
	AssertTrue(Condition := fb.dec >= -90.0 AND fb.dec <= 90.0 AND fb.ra >= 0.0 AND fb.ra < 360.0, Message := 'observer at 28.3 deg');
END_FOR
TEST_FINISHED();
END_METHOD

METHOD PRIVATE Azimuth_Difference_Is_Not_A_Sky_Separation
VAR
	fb1	: AstroBROT.FB_EQ2HOR;
	fb2	: AstroBROT.FB_EQ2HOR;
	fAzDiff	: LREAL;
END_VAR
TEST('Azimuth_Difference_Is_Not_A_Sky_Separation');
// The review recorded "azimuth outliers up to 40 arcsec" as a coordinate difference. Two positions 0.63 arcsec apart on the sky
// (0.05 deg from the zenith) differ by 629 arcsec in azimuth: the azimuth difference is amplified by 1 / cos(alt) = 1146.
// A raw azimuth difference therefore cannot be used as an accuracy figure; a great-circle separation can.
fb1(ra := 69.29947685614172, dec := 28.289165400359746, jd := 2461300.75, lon := -16.5, lat := 28.3, refract := FALSE);
fb2(ra := 69.29967685614173, dec := 28.289165400359746, jd := 2461300.75, lon := -16.5, lat := 28.3, refract := FALSE);
fAzDiff := fb2.az - fb1.az;
CheckNear(0.17470443800883118, fAzDiff, 1.0E-6, 'azimuth difference in degrees');
CheckSeparation(fb1.az, fb1.alt, fb2.az, fb2.alt, 0.00017709654618499777, 'separation of the two outputs is the sky separation');
AssertTrue(Condition := ABS(fAzDiff) > 100.0 * 0.00017609654618499777, Message := 'the azimuth difference is more than 100 times the separation');
TEST_FINISHED();
END_METHOD

END_FUNCTION_BLOCK

// ---- POUs/MAIN.TcPOU
PROGRAM MAIN
VAR
	// TcUnit finds every FB_TestSuite instance by itself; it is enough to declare them here.
	fbEq2HorTests	: FB_EQ2HOR_Tests;
	fbHor2EqTests	: FB_HOR2EQ_Tests;
	fbCoRefractTests	: FB_CO_REFRACT_Tests;
	fbCoAberrationTests	: FB_CO_ABERRATION_Tests;
	fbCoNutateTests	: FB_CO_NUTATE_Tests;
	fbTenTests	: FB_TEN_Tests;
	fbAltaz2HadecTests	: FB_ALTAZ2HADEC_Tests;
	fbAtan2Tests	: FB_ATAN2_Tests;
	fbDateTime2JdTests	: FB_DateTime2JD_Tests;
	fbJd2LstTests	: FB_JD2LST_Tests;
	fbDut1Tests	: FB_DUT1_Tests;
	fbPrecessTests	: FB_PRECESS_Tests;
	fbRadec2HadecTests	: FB_RADEC2HADEC_Tests;
	fbHadec2RadecTests	: FB_HADEC2RADEC_Tests;
	fbSunposTests	: FB_SUNPOS_Tests;
	fbEdgeCasesTests	: FB_EdgeCases_Tests;
	fbPipelineTests	: FB_Pipeline_Tests;
END_VAR

TcUnit.RUN();

END_PROGRAM
